(* LS Electric XG5000 project: Coffee_make *)
(* PLC LSPLC *)

PROGRAM NewProgram (* task: 스캔 프로그램 *)
VAR
    다음으로 : BOOL;
    다음으로자가유지 : BOOL;
    물끓이기 : TON;
    물무게 AT %MW11 : INT;
    물무게UDINT : UDINT;
    물무게곱하기 : INT;
    물투입 : TON;
    물투입시간 : TIME;
    물투입통과 : BOOL;
    섞기 : TON;
    섞기통과 : BOOL;
    시럽무게곱하기 : INT;
    시럽우유무게UDINT : UDINT;
    시럽우유투입 : TON;
    시럽우유투입시간 : TIME;
    얼음선투입 AT %MX16 : BOOL;
    얼음선투입타이머 : TON;
    얼음선투입통과 : BOOL;
    얼음후투입 AT %MX17 : BOOL;
    얼음후투입타이머 : TON;
    얼음후투입통과 : BOOL;
    에이드액무게 : INT := 0;
    에이드투입 : BOOL := 0;
    우유뎁히기 : TON;
    우유무게 AT %MW12 : INT := 0;
    우유무게UDINT : UDINT;
    우유무게곱하기 : INT;
    우유투입 : TON;
    우유투입시간 : TIME;
    우유투입여부 : BOOL;
    우유투입통과 : BOOL;
    원두갈기 : TON;
    원두넣기 : TON;
    원두넣기시간 : TIME := T#5s;
    원두추출 : TON;
    음료제조시작 AT %IX0.0.1 : BOOL;
    음료제조완료 AT %QX0.1.0 : BOOL;
    음료제조자가유지 : BOOL;
    일단멈춰 : BOOL := 0;
    일단멈춰2 : BOOL;
    일단멈춰3 : BOOL;
    일단멈춰4 : BOOL;
    일단멈춰5 : BOOL;
    일단멈춰6 : BOOL;
    일단멈춰7 : BOOL;
    일단멈춰8 : BOOL;
    초코시럽무게 AT %MW13 : INT;
    초코시럽무게UDINT : UDINT;
    초코시럽무게곱하기 : INT;
    초코시럽투입 : TON;
    초코시럽투입시간 : TIME;
    초코시럽투입여부 : BOOL;
    초코시럽투입통과 : BOOL;
    카페시럽무게 AT %MW14 : INT := 0;
    카페시럽무게UDINT : UDINT;
    카페시럽무게곱하기 : INT;
    카페시럽투입 : TON;
    카페시럽투입1 : TON;
    카페시럽투입2 : TON;
    카페시럽투입시간 : TIME;
    카페시럽투입여부 : BOOL;
    카페시럽투입통과 : BOOL;
    커피가레일로 : TON;
    커피끓이기시간 : TIME;
    커피무게 AT %MW10 : INT;
    커피무게UDINT : UDINT;
    커피무게곱하기 : INT;
    커피온도 AT %MW15 : INT;
    커피온도UDINT : UDINT;
    커피온도곱하기 : INT;
    커피추출 : TON;
    커피투입 : TON;
    커피투입시간 : TIME;
    커피투입시작 : BOOL;
    커피투입통과 : BOOL;
    컵구멍인지 : TON;
    컵투입 : TON;
    컵투입통과 : BOOL;
    호퍼닫기 : BOOL;
END_VAR
VAR
    _t1 : BOOL;
    _t2 : BOOL;
    _p3 : BOOL;
    _t4 : BOOL;
END_VAR

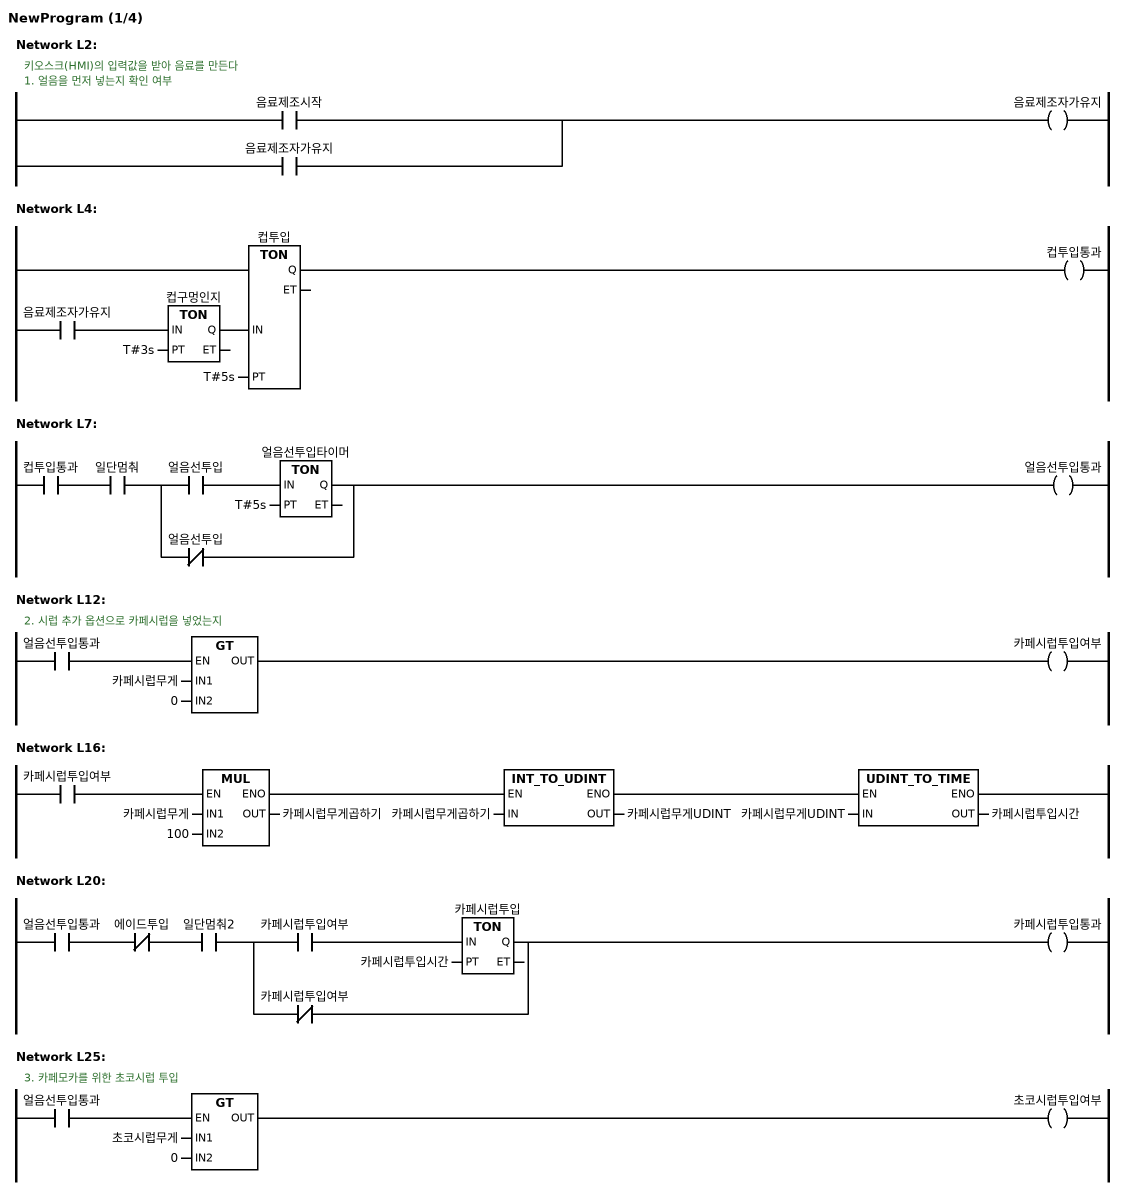
(* 키오스크(HMI)의 입력값을 받아 음료를 만든다 *)
(* 1. 얼음을 먼저 넣는지 확인 여부 *)
(* Rung L2 *)
음료제조자가유지 := 음료제조시작 OR 음료제조자가유지;
(* Rung L4 *)
컵구멍인지(IN := 음료제조자가유지, PT := T#3s);
컵투입(IN := 컵구멍인지.Q, PT := T#5s);
컵투입통과 := 컵투입.Q;
(* Rung L7 *)
얼음선투입타이머(IN := 컵투입통과 AND 일단멈춰 AND 얼음선투입, PT := T#5s);
얼음선투입통과 := 얼음선투입타이머.Q OR (컵투입통과 AND 일단멈춰 AND NOT 얼음선투입);
(* 2. 시럽 추가 옵션으로 카페시럽을 넣었는지 *)
(* Rung L12 *)
IF 얼음선투입통과 THEN _t1 := 카페시럽무게 > 0; END_IF;
카페시럽투입여부 := _t1;
(* Rung L16 *)
IF 카페시럽투입여부 THEN
    카페시럽무게곱하기 := 카페시럽무게 * 100;
    카페시럽무게UDINT := INT_TO_UDINT(카페시럽무게곱하기);
    카페시럽투입시간 := UDINT_TO_TIME(카페시럽무게UDINT);
END_IF;
(* Rung L20 *)
카페시럽투입(IN := 얼음선투입통과 AND NOT 에이드투입 AND 일단멈춰2 AND 카페시럽투입여부, PT := 카페시럽투입시간);
카페시럽투입통과 := 카페시럽투입.Q OR (얼음선투입통과 AND NOT 에이드투입 AND 일단멈춰2 AND NOT 카페시럽투입여부);
(* 3. 카페모카를 위한 초코시럽 투입 *)
(* Rung L25 *)
IF 얼음선투입통과 THEN _t2 := 초코시럽무게 > 0; END_IF;
초코시럽투입여부 := _t2;

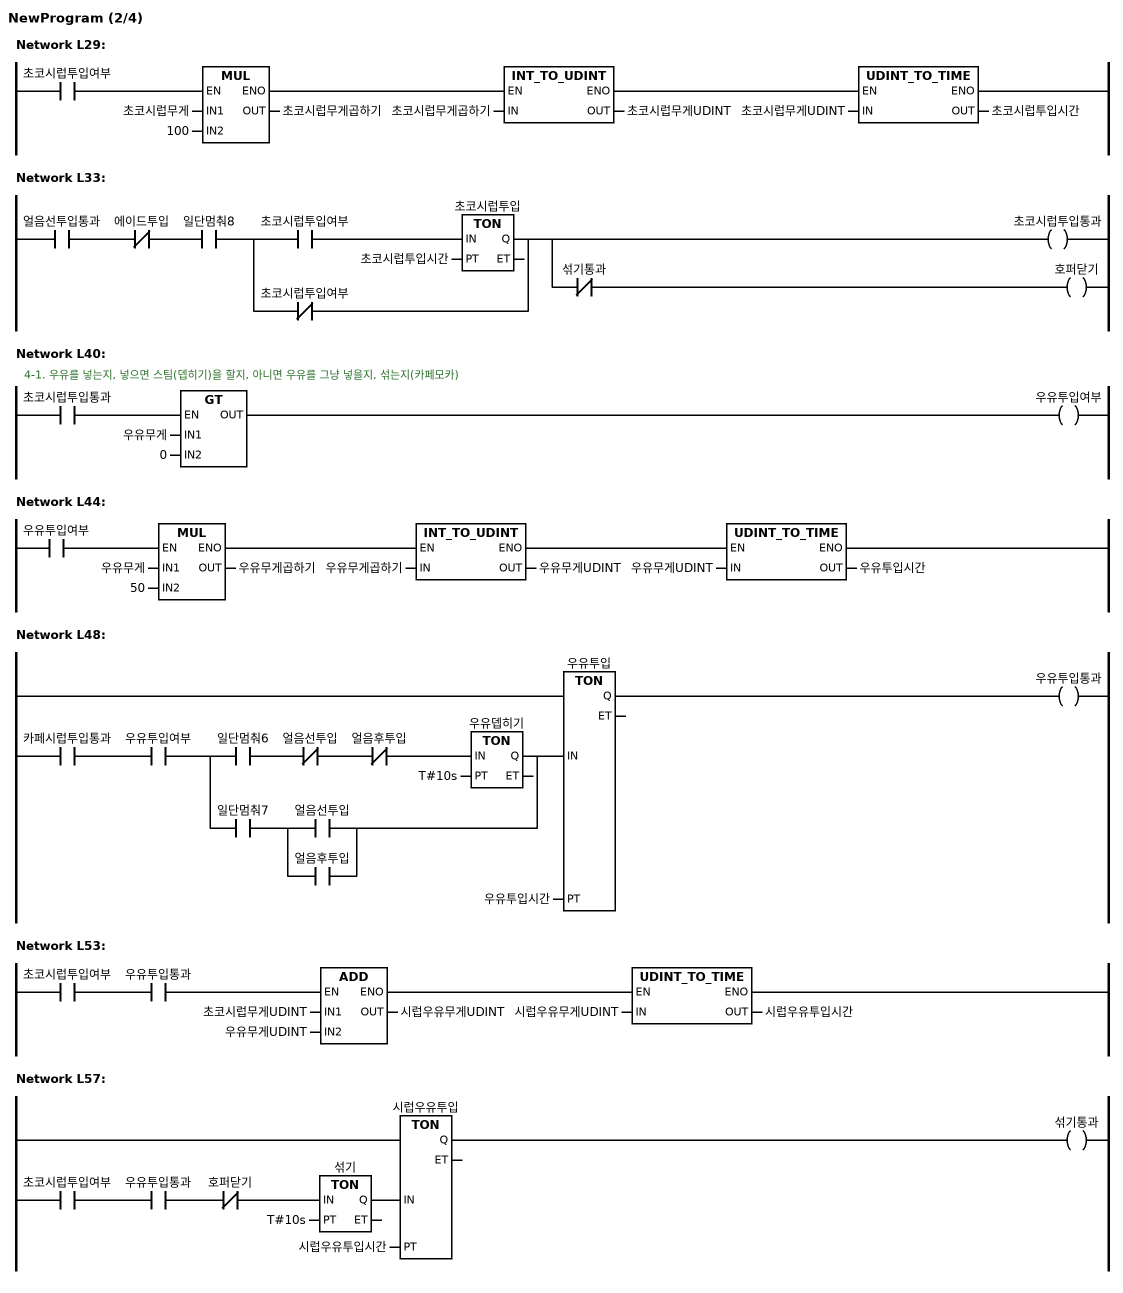
(* Rung L29 *)
IF 초코시럽투입여부 THEN
    초코시럽무게곱하기 := 초코시럽무게 * 100;
    초코시럽무게UDINT := INT_TO_UDINT(초코시럽무게곱하기);
    초코시럽투입시간 := UDINT_TO_TIME(초코시럽무게UDINT);
END_IF;
(* Rung L33 *)
초코시럽투입(IN := 얼음선투입통과 AND NOT 에이드투입 AND 일단멈춰8 AND 초코시럽투입여부, PT := 초코시럽투입시간);
_p3 := 초코시럽투입.Q OR (얼음선투입통과 AND NOT 에이드투입 AND 일단멈춰8 AND NOT 초코시럽투입여부);
초코시럽투입통과 := _p3;
호퍼닫기 := _p3 AND NOT 섞기통과;
(* 4-1. 우유를 넣는지, 넣으면 스팀(뎁히기)을 할지, 아니면 우유를 그냥 넣을지, 섞는지(카페모카) *)
(* Rung L40 *)
IF 초코시럽투입통과 THEN _t4 := 우유무게 > 0; END_IF;
우유투입여부 := _t4;
(* Rung L44 *)
IF 우유투입여부 THEN
    우유무게곱하기 := 우유무게 * 50;
    우유무게UDINT := INT_TO_UDINT(우유무게곱하기);
    우유투입시간 := UDINT_TO_TIME(우유무게UDINT);
END_IF;
(* Rung L48 *)
우유뎁히기(IN := 카페시럽투입통과 AND 우유투입여부 AND 일단멈춰6 AND NOT 얼음선투입 AND NOT 얼음후투입, PT := T#10s);
우유투입(IN := 우유뎁히기.Q OR (카페시럽투입통과 AND 우유투입여부 AND 일단멈춰7 AND (얼음선투입 OR 얼음후투입)), PT := 우유투입시간);
우유투입통과 := 우유투입.Q;
(* Rung L53 *)
IF 초코시럽투입여부 AND 우유투입통과 THEN
    시럽우유무게UDINT := 초코시럽무게UDINT + 우유무게UDINT;
    시럽우유투입시간 := UDINT_TO_TIME(시럽우유무게UDINT);
END_IF;
(* Rung L57 *)
섞기(IN := 초코시럽투입여부 AND 우유투입통과 AND NOT 호퍼닫기, PT := T#10s);
시럽우유투입(IN := 섞기.Q, PT := 시럽우유투입시간);
섞기통과 := 시럽우유투입.Q;

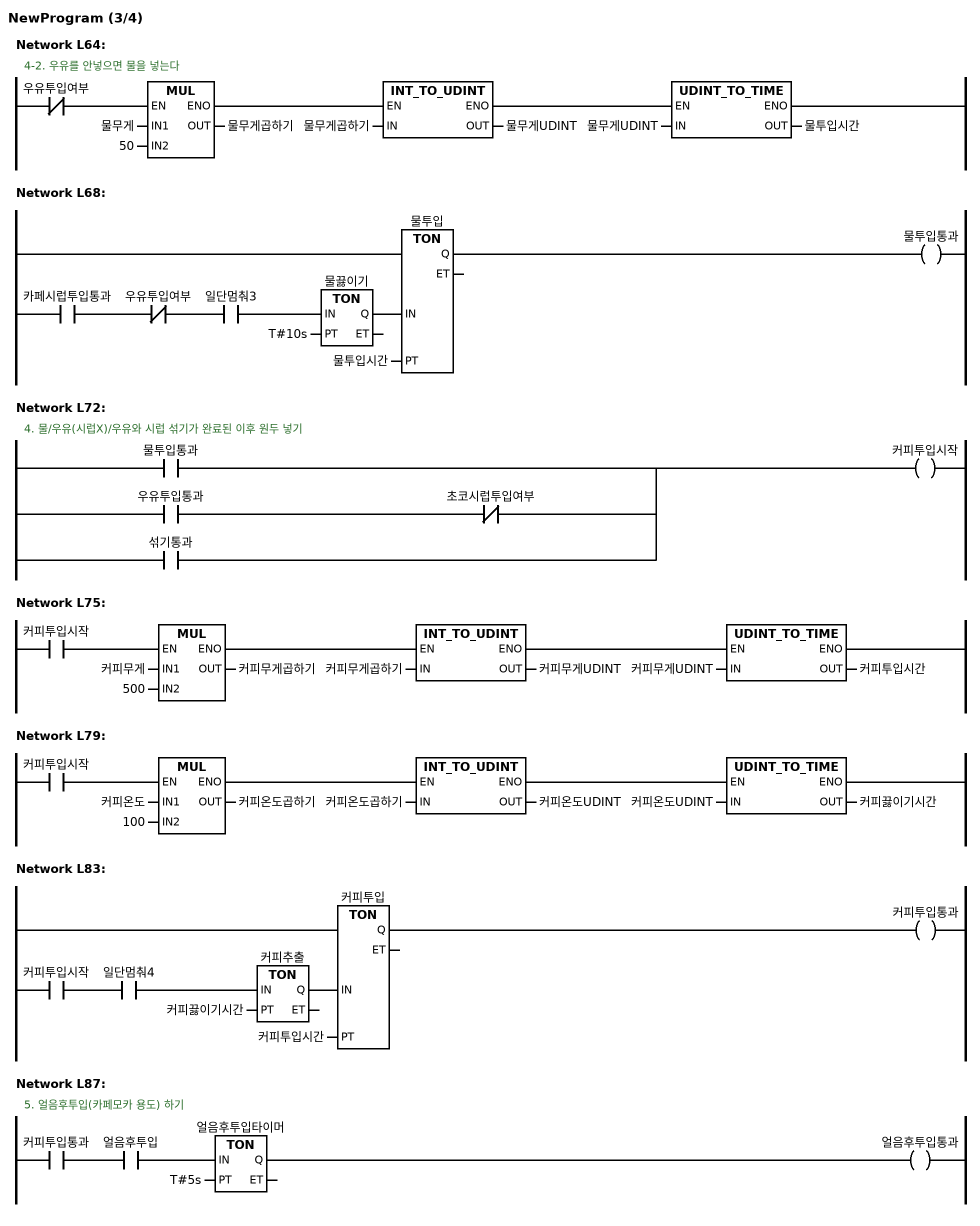
(* 4-2. 우유를 안넣으면 물을 넣는다 *)
(* Rung L64 *)
IF NOT 우유투입여부 THEN
    물무게곱하기 := 물무게 * 50;
    물무게UDINT := INT_TO_UDINT(물무게곱하기);
    물투입시간 := UDINT_TO_TIME(물무게UDINT);
END_IF;
(* Rung L68 *)
물끓이기(IN := 카페시럽투입통과 AND NOT 우유투입여부 AND 일단멈춰3, PT := T#10s);
물투입(IN := 물끓이기.Q, PT := 물투입시간);
물투입통과 := 물투입.Q;
(* 4. 물/우유(시럽X)/우유와 시럽 섞기가 완료된 이후 원두 넣기 *)
(* Rung L72 *)
커피투입시작 := 물투입통과 OR (우유투입통과 AND NOT 초코시럽투입여부) OR 섞기통과;
(* Rung L75 *)
IF 커피투입시작 THEN
    커피무게곱하기 := 커피무게 * 500;
    커피무게UDINT := INT_TO_UDINT(커피무게곱하기);
    커피투입시간 := UDINT_TO_TIME(커피무게UDINT);
END_IF;
(* Rung L79 *)
IF 커피투입시작 THEN
    커피온도곱하기 := 커피온도 * 100;
    커피온도UDINT := INT_TO_UDINT(커피온도곱하기);
    커피끓이기시간 := UDINT_TO_TIME(커피온도UDINT);
END_IF;
(* Rung L83 *)
커피추출(IN := 커피투입시작 AND 일단멈춰4, PT := 커피끓이기시간);
커피투입(IN := 커피추출.Q, PT := 커피투입시간);
커피투입통과 := 커피투입.Q;
(* 5. 얼음후투입(카페모카 용도) 하기 *)
(* Rung L87 *)
얼음후투입타이머(IN := 커피투입통과 AND 얼음후투입, PT := T#5s);
얼음후투입통과 := 얼음후투입타이머.Q;

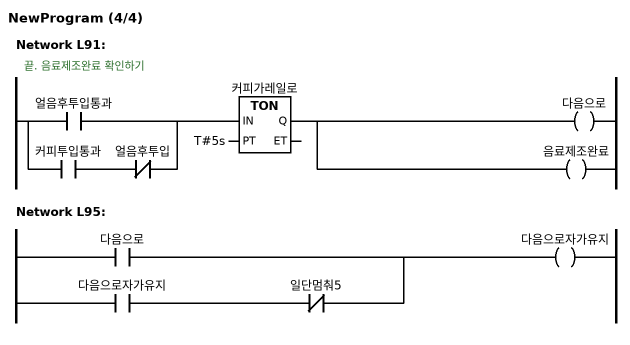
(* 끝. 음료제조완료 확인하기 *)
(* Rung L91 *)
커피가레일로(IN := 얼음후투입통과 OR (커피투입통과 AND NOT 얼음후투입), PT := T#5s);
다음으로 := 커피가레일로.Q;
음료제조완료 := 커피가레일로.Q;
(* Rung L95 *)
다음으로자가유지 := 다음으로 OR (다음으로자가유지 AND NOT 일단멈춰5);
END_PROGRAM